FUNCTION FC_WIDP_TO_PPNAME : STRING
VAR_INPUT
	WindP					: STRING;
END_VAR
VAR
	i				: INT;
	tempPPINT 		: INT;
	tempPPString	: STRING;
END_VAR

tempPPINT := LEN(WindP);
tempPPString := WindP;
IF tempPPINT < 8 THEN
	FOR i := 0 TO 7-tempPPINT DO
		tempPPString := CONCAT('0', tempPPString);
	END_FOR
END_IF
FC_WIDP_TO_PPNAME := tempPPString;

END_FUNCTION

(* stored: Version 1.1.0.1, ProductVersion 3.1.4024.13
   POU FC_WIDP_TO_PPNAME: Id {d8e4615f-037f-4e79-8ccd-408226bbabc5}, SpecialFunc None *)
